// TIA Portal V17 export
// export: Created 2025-03-12T14:52:36.9050991Z, ExportSetting WithDefaults, DisplayName Totally Integrated Automation Portal, DisplayVersion V17 Update 8, DisplayName TIA Portal Openness, DisplayVersion V17 Update 8, DisplayName TIA Portal Version Control Interface, DisplayVersion V17, DisplayName SINAMICS Startdrive Advanced, DisplayVersion V17 SP2, DisplayName SINAMICS Startdrive G110M, G120, G120C, G120D, G120P, G115D, DisplayVersion V17 SP2, DisplayName SINAMICS Startdrive G130, G150, S120, S150, SINAMICS MV, S210, DisplayVersion V17 SP2, DisplayName STEP 7 Professional, DisplayVersion V17 Update 8, DisplayName SINUMERIK ONE STEP 7 Toolbox, DisplayVersion V17 Update 12, DisplayName SINUMERIK 840D sl STEP 7 Toolbox, DisplayVersion V17 Update 12, DisplayName STEP 7 Safety, DisplayVersion V17 Update 6, DisplayName WinCC Advanced, DisplayVersion V17 Update 8
TYPE "POWDER FEEDER HMI ACTIONS"
// stored: IsFailsafeCompliant false
   STRUCT
      SWITCH_ON_HEATER_LINE_1 : Bool;   // SWITCH ON HEATER LINE 1 HMI REQUEST
      SWITCH_OFF_HEATER_LINE_1 : Bool;   // SWITCH OFF HEATER LINE 1 HMI REQUEST
      SWITCHED_ON_HEATER_LINE_1 : Bool;   // SWITCHED ON HEATER LINE 1 HMI STATUS
      SWITCHED_OFF_HEATER_LINE_1 : Bool;   // SWITCHED OFF HEATER LINE 1 HMI STATUS
      SWITCH_ON_HEATER_LINE_2 : Bool;   // SWITCH ON HEATER LINE 2 HMI REQUEST
      SWITCH_OFF_HEATER_LINE_2 : Bool;   // SWITCH OFF HEATER LINE 2 HMI REQUEST
      SWITCHED_ON_HEATER_LINE_2 : Bool;   // SWITCHED ON HEATER LINE 2 HMI STATUS
      SWITCHED_OFF_HEATER_LINE_2 : Bool;   // SWITCHED OFF HEATER LINE 2 HMI STATUS
      SWITCH_ON_HOOPER_LINE_1 : Bool;   // SWITCH ON HOOPER LINE 1 HMI REQUEST
      SWITCH_OFF_HOOPER_LINE_1 : Bool;   // SWITCH OFF HOOPER LINE 1 HMI REQUEST
      SWITCHED_ON_HOOPER_LINE_1 : Bool;   // SWITCHED ON HOOPER LINE 1 HMI STATUS
      SWITCHED_OFF_HOOPER_LINE_1 : Bool;   // SWITCHED OFF HOOPER LINE 1 HMI STATUS
      SWITCH_ON_HOOPER_LINE_2 : Bool;   // SWITCH ON HOOPER LINE 2 HMI REQUEST
      SWITCH_OFF_HOOPER_LINE_2 : Bool;   // SWITCH OFF HOOPER LINE 2 HMI REQUEST
      SWITCHED_ON_HOOPER_LINE_2 : Bool;   // SWITCHED ON HOOPER LINE 2 HMI STATUS
      SWITCHED_OFF_HOOPER_LINE_2 : Bool;   // SWITCHED OFF HOOPER LINE 2 HMI STATUS
      SELECT_ARGON_GAS : Bool;   // SELECT ARGON GAS HMI REQUEST
      SELECT_NITROGEN_GAS : Bool;   // SELECT NITROGEN GAS HMI REQUEST
      SELECT_HELIUM_GAS : Bool;   // SELECT HELIUM GAS HMI REQUEST
      SELECT_ARGON30_GAS : Bool;   // SELECT ARGON30 GAS HMI REQUEST
      SELECTED_ARGON_GAS : Bool;   // SELECTED ARGON GAS HMI STATUS
      SELECTED_NITROGEN_GAS : Bool;   // SELECTED NITROGEN GAS HMI STATUS
      SELECTED_HELIUM_GAS : Bool;   // SELECTED HELIJM GAS HMI STATUS
      SELECTED_ARGON30_GAS : Bool;   // SELECTED ARGON30 GAS HMI STATUS
      SELECT_METRIC_UNITS : Bool;   // SELECT METRIC UNITS HMI REQUEST
      SELECT_IMPERIAL_UNITS : Bool;   // SELECT IMPERIAL UNITS HMI REQUEST
      SELECTED_METRIC_UNITS : Bool;   // SELECTED METRIC UNITS HMI STATUS
      SELECTED_IMPERIAL_UNITS : Bool;   // SELECTED IMPERIAL UNITS HMI STATUS
   END_STRUCT;
END_TYPE
